(* CoDeSys 2.3.9.42 project: CR0403 AGV_25.pro *)
(* Libraries: SysLibVisu.lib 16.9.03 13:17:00, SysLibPlcCtrl.lib 13.6.03 15:49:00, SysLibFile.lib 23.9.04 10:11:36, SysLibTime.lib 27.4.05 10:36:52, SysLibTargetVisu.lib 5.4.04 13:31:00, LinuxSystemLib.Lib 18.3.03 13:26:50, ifm_CANopen\ifm_CANopen_NT_V020004.lib 3.11.15 19:07:50, ifm_pdm_file_V010006.lib 14.1.08 14:21:32, ifm_CR0403\ifm_CR0403_V030100.lib 15.1.16 15:49:16, Util.lib 6.11.07 16:39:24, ifm_J1939_NT\ifm_J1939_NT_V020004.lib 18.9.14 16:13:02, ifm_RAWCan\ifm_RAWCan_NT_V020004.lib 3.11.15 19:07:52, standard.lib 4.10.05 12:14:46, SysLibCallback.lib 26.9.08 17:43:52 *)

(* PLC configuration (modules and I/O channels)
Configuration [LocalConfiguration] node 0, in %IB0 out %QB0 {IFM_PARAM_WORD_TIME = 0}
Input/Output [LocalInputOutput] node 1, in %IB0 out %QB0
  Inputs Binary [LocalIn] node 0, in %IB0 out %QB0
    IN00 AT %IB0 [ChInputBool] Input 00 Bit
    IN01 AT %IB1 [ChInputBool] Input 01 Bit
    IN02 AT %IB2 [ChInputBool] Input 02 Bit
    IN03 AT %IB3 [ChInputBool] Input 03 Bit
    IN04 AT %IB4 [ChInputBool] Input 04 Bit
    IN05 AT %IB5 [ChInputBool] Input 05 Bit
    IN06 AT %IB6 [ChInputBool] Input 06 Bit
    IN07 AT %IB7 [ChInputBool] Input 07 Bit
    IN08 AT %IB8 [ChInputBool] Input 08 Bit
    IN09 AT %IB9 [ChInputBool] Input 09 Bit
    IN10 AT %IB10 [ChInputBool] Input 10 Bit
    IN11 AT %IB11 [ChInputBool] Input 11 Bit
  Outputs Binary [LocalOut] node 1, in %IB12 out %QB0
    OUT00 AT %QB0 [ChOutputBool] Output 00 Bit
    OUT01 AT %QB1 [ChOutputBool] Output 01 Bit
    OUT02 AT %QB2 [ChOutputBool] Output 02 Bit
    OUT03 AT %QB3 [ChOutputBool] Output 03 Bit
    OUT04 AT %QB4 [ChOutputBool] Output 04 Bit
    OUT05 AT %QB5 [ChOutputBool] Output 05 Bit
    OUT06 AT %QB6 [ChOutputBool] Output 06 Bit
    OUT07 AT %QB7 [ChOutputBool] Output 07 Bit
    OUT08 AT %QB8 [ChOutputBool] Output 08 Bit
    OUT09 AT %QB9 [ChOutputBool] Output 09 Bit
    OUT10 AT %QB10 [ChOutputBool] Output 10 Bit
    OUT11 AT %QB11 [ChOutputBool] Output 11 Bit
  System Inputs [LocalSystemInputs] node 2, in %IB12 out %QB12
    SUPPLY_VOLTAGE_VBBS AT %IW6 [ChInputWord] Supply voltage VBBS
    SUPPLY_VOLTAGE_VU AT %IW7 [ChInputWord] Supply voltage VU
    SUPPLY_VOLTAGE_VBB1 AT %IW8 [ChInputWord] Supply voltage VBB1
    SUPPLY_VOLTAGE_VBB2 AT %IW9 [ChInputWord] Supply voltage VBB2
    TEMPERATURE AT %IW10 [ChInputInt] Temperature
J1939 Interface [CAN_J1939] node 1, in %IB60 out %QB44
J1939 Interface [CAN_J1939] node 1, in %IB76 out %QB76
*)

(* Global variable list: Global_Variables *)
VAR_GLOBAL
	Route1: ARRAY [1..2,1..4] OF REAL := 10, 100, 100, 10, 10, 10, 100, 100;
	(*Route1: ARRAY [1..2,1..4] OF REAL := 10, 60, 140, 10, 10, 30, 30, 130;*)


END_VAR

VAR_GLOBAL RETAIN	(*Onze array die de aangeleerde route bevat moet een RETAIN variable zijn opdat deze zijn waarden zou blijven kennen ook bij afzetten van de spanning*)
	RouteLeren: ARRAY [1..2, 1..10] OF DWORD;
END_VAR

(* Data type *)
TYPE CONSTANTS_MATH :
STRUCT
	RadDeg : REAL := 57.29577951; (*Conversie van radialen naar degrees*)
	PI : REAL := 	3.14159265358979323846264338327950288;		(* Kreiszahl PI *)
	PI2 : REAL := 	6.28318530717958647692528676655900576;	(* PI * 2 *)
	PI4 : REAL :=  12.56637061435917295385057353311801152;	(* PI * 4 *)
	PI05 : REAL :=  1.5707963267949;							(* PI / 2 *)
	PI025 : REAL := 0.785398163397448;							(* PI / 4 *)
	PI_INV : REAL := 0.318309886183791;						(* 1 / PI *)
	E : REAL := 	2.71828182845904523536028747135266249;		(* Euler constant e *)
	E_INV : REAL := 0.367879441171442;							(* 1 / e *)
	SQ2 : REAL :=	1.4142135623731;							(* Wurzel von 2 *)
	FACTS : ARRAY[0..12] OF DINT := 1,1,2,6,24,120,720,5040,40320,362880,3628800,39916800,479001600;
END_STRUCT
END_TYPE

(* POU PLC_PRG, ST *)
PROGRAM PLC_PRG
VAR
	CAN_ENABLE_CAN2: CAN_ENABLE;
	CAN_ENABLE_CAN1: CAN_ENABLE;

	CAN_RX_ModusAGV: CAN_RX;
	Manueel: BOOL;
	Leren: BOOL;
	Automatisch: BOOL;
	UNPACK_ModusAGV: UNPACK;
	test1: BOOL;
	test2: BOOL;
END_VAR
(*Enabelen van CAN bus 1*)
CAN_ENABLE_CAN1(
	ENABLE:=TRUE ,
	CHANNEL:=1 ,
	BAUDRATE:=500 ,
	RESULT=> );

(*Enabelen van CAN bus 2 voor hetronic*)
CAN_ENABLE_CAN2(
	ENABLE:=TRUE ,
	CHANNEL:=2 ,
	BAUDRATE:=125 ,
	RESULT=> );

(*Binnenlezen modus AGV*)
CAN_RX_ModusAGV(
	ENABLE				:= TRUE,
	CHANNEL				:=1 ,
	ID						:= 16#191,
	DATA					=> ,
	RESULT				=> );

IF CAN_RX_ModusAGV.RESULT = 1
THEN
	UNPACK_ModusAGV(
	B:= CAN_RX_ModusAGV.DATA[0] ,
	B0=>Manueel ,
	B1=>Leren,
	B2=>Automatisch ,
	B3=> , 
	B4=> ,
	B5=> , 
	B6=> , 
	B7=> );
END_IF

(*Programma's die continu moeten uitgevoerd worden ongeacht de modus*)
VoedingContactor();
CAN_RX_comm_display();

(*Afhankelijk van de gewenste modus voeren we één van de onderstaande programma's uit*)
IF Manueel = TRUE
THEN
ManueleBediening();
ELSIF Leren = TRUE
THEN
AanlerenRoute();
ELSIF Automatisch = TRUE
THEN
NavSof();
END_IF
END_PROGRAM

(* POU VoedingContactor, ST *)
PROGRAM VoedingContactor
VAR

	PWM1000_Contactor_OUT7: PWM1000;
	wContactor_voeding: WORD;
	bContactor_voeding: BYTE;
END_VAR
PWM1000_Contactor_OUT7(
	ENABLE:=						TRUE ,
	CHANNEL:=					7 ,
	FREQUENCY:=				100 ,
	VALUE:=						1000 ,
	DITHER_FREQUENCY:= ,
	DITHER_VALUE:= , 
	CURRENT=>					wContactor_voeding,
	RESULT=> 					bContactor_voeding);
END_PROGRAM

(* POU CAN_RX_comm_display, ST *)
PROGRAM CAN_RX_comm_display
VAR
	CAN_RX_comm_keys_display: CAN_RX;
	UNPACK_comm_keys: UNPACK;
	keyF1: BOOL;
	keyF2: BOOL;
	keyF3: BOOL;
	keyF4: BOOL;
END_VAR
CAN_RX_comm_keys_display(
	ENABLE:=TRUE ,
	CHANNEL:=1 ,
	ID:=16#190 ,
	DATA=> ,
	RESULT=> );

IF CAN_RX_comm_keys_display.RESULT=1  THEN

UNPACK_comm_keys(
	B:=CAN_RX_comm_keys_display.DATA[0] ,
	B0=>keyF1 ,
	B1=>keyF2 ,
	B2=>keyF3,
	B3=>keyF4 ,
	B4=> ,
	B5=> , 
	B6=> , 
	B7=> );


END_IF

IF keyF1 THEN
OUT00:=TRUE;
ELSE
OUT00:=FALSE;
END_IF

IF keyF2 THEN
OUT01:=TRUE;
ELSE
OUT01:=FALSE;
END_IF
END_PROGRAM

(* POU ManueleBediening, ST *)
PROGRAM ManueleBediening
VAR
	(*Binnenlezen as1  APEM HFX*)
	INPUT_IN01_Voor_achter: INPUT;
	wVoorAchter: WORD;
	bVoorAchter: BYTE;

	(*Binnenlezen as2  APEM HFX*)
	INPUT_IN00_Links_Rechts: INPUT;
	wLinksRechts: WORD;
	bLinksRechts: BYTE;

	(*Variabele waarin de gewenste richting en snelheid wordt weggeschreven*)
	wSnelheid_ch1: DWORD := 0;
	wSnelheid_ch2: DWORD := 0;

	(*Frequentie waarop SDO write bericht verzonden wordt*)
	BLINK_SDOBericht: BLINK;
	xSDO: BOOL;

	(*SDO bericht voor channel 1 en channel 2*)
	CANOPEN_SDOWRITE_ManueleBediening_ch1: CANOPEN_SDOWRITE;
	CANOPEN_SDOWRITE_ManueleBediening_ch2: CANOPEN_SDOWRITE;
	DWORD_TO_ARRAY_ch1: DWORD_TO_ARRAY;
	DWORD_TO_ARRAY_ch2: DWORD_TO_ARRAY;

	X_as_hetronic: WORD;
	Y_as_hetronic: WORD;
	rSnelheid_ch1: REAL;
	rSnelheid_ch2: REAL;
END_VAR
(*Hier moeten we de APEM HFX binnenlezen
- Blauwe draad (verbinden we met IN01 van de CR0403:
	- Vooruit (2.5V --> 4.7V)
	- Achteruit (2.5V --> 0V)
- Gele draad (verbinden we met IN00 van de CR0403):
	- Links (2.5 --> 4.7V)
	- Rechts (2.5V --> 0V)
De switch bovenop de joystick verbindt de witte draad en de oranje draad bij indrukken
==> Deze willen we gebruiken om coördinaten op te slaan*)
(*INPUT FB om waarden as 1 joystick binnen te lezen*)
	(*INPUT_IN01_Voor_achter(
		ENABLE				:= TRUE,
		CHANNEL				:= 1,					(*We gebruiken IN01*)
		MODE					:= 3,					(*Voltage input 0 ... 10000 mV*)
		FILTER				:= ,
		VALUE					=> wVoorAchter ,		(*Bevat de spanningswaarde die we binnenlezen op IN00*)
		RESULT				=>bVoorAchter );		(*Als deze op 1 staat wil dat zeggen dat de FB is executed without error*)
(*INPUT FB om waarden as 2 joystick binnen te lezen*)
	INPUT_IN00_Links_Rechts(
		ENABLE				:= TRUE,
		CHANNEL				:= 0,					(*We gebruiken IN01*)
		MODE					:= 3,					(*Voltage input 0 ... 10000 mV*)
		FILTER				:= ,
		VALUE					=> wLinksRechts ,		(*Bevat de spanningswaarde die we binnenlezen op IN00*)
		RESULT				=>bLinksRechts );*)	(*Als deze op 1 staat wil dat zeggen dat de FB is executed without error*)

X_as_hetronic := X_as;
Y_as_hetronic := Y_as;


(*Frequentie waarop ons SDO bericht voor de roboteq aan te sturen op de bus geplaatst wordt*)
BLINK_SDOBericht(
ENABLE:= TRUE ,
TIMELOW:= t#10ms,
TIMEHIGH:=t#10ms ,
OUT=> xSDO );

(*Channel 1 Roboteq SDC2130*)
CANOPEN_SDOWRITE_ManueleBediening_ch1(
	EXECUTE				:= xSDO,
	CHANNEL				:= 1,
	NODE					:=2 ,
	IDX						:=16#2000,
	SUBIDX				:= 16#1,
	LEN					:=4 ,
	DATA					:= ,
	Timeout				:= ,
	RESULT				=> );

DWORD_TO_ARRAY_ch1(
	Word_In:=wSnelheid_ch1 ,
	P_0=>CANOPEN_SDOWRITE_ManueleBediening_ch1.DATA[0] ,
	P_1=>CANOPEN_SDOWRITE_ManueleBediening_ch1.DATA[1] ,
	P_2=>CANOPEN_SDOWRITE_ManueleBediening_ch1.DATA[2] ,
	P_3=>CANOPEN_SDOWRITE_ManueleBediening_ch1.DATA[3] );

(*Channel 2 Roboteq SDC2130*)
CANOPEN_SDOWRITE_ManueleBediening_ch2(
	EXECUTE				:= xSDO,
	CHANNEL				:= 1,
	NODE					:=2 ,
	IDX						:=16#2000,
	SUBIDX				:= 16#2,
	LEN					:=4 ,
	DATA					:= ,
	Timeout				:= ,
	RESULT				=> );

DWORD_TO_ARRAY_ch2(
	Word_In:=wSnelheid_ch2,
	P_0=>CANOPEN_SDOWRITE_ManueleBediening_ch2.DATA[0] ,
	P_1=>CANOPEN_SDOWRITE_ManueleBediening_ch2.DATA[1] ,
	P_2=>CANOPEN_SDOWRITE_ManueleBediening_ch2.DATA[2] ,
	P_3=>CANOPEN_SDOWRITE_ManueleBediening_ch2.DATA[3] );










(*VOOR_ACHTER: Vooruit en achteruit rijden*)
IF Y_as < 126 	AND X_as = 127
THEN
	(*Vooruitrijden (onderstaande commands zorgen ervoor dat onze differential drive robot rechtuit rijdt)*)
		wSnelheid_ch1 := (0+ (10*(127 - Y_as)));
		wSnelheid_ch2 := (65536 - (10*(127 - Y_as)));

ELSIF

Y_as > 128 AND X_as = 127
THEN
	(*Achteruitrijden (onderstaande commands zorgen ervoor dat onze differential drive robot rechtuit naar achter rijdt)*)
		wSnelheid_ch1 :=(65536 + (10*(127 - Y_as)));
		wSnelheid_ch2 := (0- (10*(127 - Y_as)));
ELSIF

(**)
X_as < 126 AND Y_as = 127
THEN
	(*Vooruitrijden (onderstaande commands zorgen ervoor dat onze differential drive robot rechtuit rijdt)*)
		wSnelheid_ch1 := (65536 - (10*(127 - X_as)));
		wSnelheid_ch2 := (65536 - (10*(127 - X_as)));
ELSIF

(**)
X_as > 128 AND Y_as = 127
THEN
	(*Achteruitrijden (onderstaande commands zorgen ervoor dat onze differential drive robot rechtuit naar achter rijdt)*)
		wSnelheid_ch1 := (0 - (10*(127 - X_as)));
		wSnelheid_ch2 := (0 - (10*(127 - X_as)));

ELSIF

Y_as = 127 AND X_as = 127
THEN
		wSnelheid_ch1 :=0;
		wSnelheid_ch2 :=0;
END_IF
(*

(*LINKS_RECHTS: Links en rechts rijden*)
IF wLinksRechts > 2700 AND  wVoorAchter > 2300 AND wVoorAchter <2700
THEN
	(*Links draaien*)
		wSnelheid_ch1 := (wLinksRechts - 2700)/2;
		wSnelheid_ch2 := 65536 - ((2400 - wLinksRechts)/2);

END_IF

IF wLinksRechts < 2300 AND  wVoorAchter > 2300 AND wVoorAchter <2700
THEN
	(*Rechts draaien*)
		wSnelheid_ch1 := 65536 - ((2400 - wLinksRechts)/2);
		wSnelheid_ch2 := (wLinksRechts - 2700)/2;
END_IF

(*STOPPEN: Als de joystick in het midden staat moet de AGV stoppen d.w.z. dat de ingelezen waarde zowel op de x-as als de y-as rond de 2.5V moeten zijn*)
IF wVoorAchter > 2300 AND wVoorAchter <2700 AND wLinksRechts > 2300 AND wLinksRechts <2700
THEN
	wSnelheid_ch1 := 0;
	wSnelheid_ch2 := 0;
END_IF


*)




















(*Hier moeten we de APEM HFX binnenlezen
- Blauwe draad (verbinden we met IN01 van de CR0403:
	- Vooruit (2.5V --> 4.7V)
	- Achteruit (2.5V --> 0V)
- Gele draad (verbinden we met IN00 van de CR0403):
	- Links (2.5 --> 4.7V)
	- Rechts (2.5V --> 0V)
De switch bovenop de joystick verbindt de witte draad en de oranje draad bij indrukken
==> Deze willen we gebruiken om coördinaten op te slaan*)
(*
(*Versturen cyclisch CAN bericht dat de motordata voor de Roboteq SDC2130 bevat*)
CAN_TX_ENH_CYCLIC_Roboteq(
	ENABLE				:= TRUE,
	CHANNEL				:= 1 ,
	ID						:= 16#E1 ,
	Extended				:= FALSE ,
	DataLengthCode		:= 6,
	DATA					:= ,
	PERIOD				:= t#10ms,
	RESULT				=> );

CAN_TX_ENH_CYCLIC_Roboteq.DATA[0] := bMotorDirection_ch1; (*Kan 0 of 1 bevatten en afh daarvan draait de motor CW of CCW*)
WORD_TO_ARRAY_ch1(
	Word_In				:= wSnelheid_ch1 ,
	P_0					=>CAN_TX_ENH_CYCLIC_Roboteq.DATA[1] ,
	P_1					=>CAN_TX_ENH_CYCLIC_Roboteq.DATA[2]);

CAN_TX_ENH_CYCLIC_Roboteq.DATA[3] := bMotorDirection_ch2;
WORD_TO_ARRAY_ch2(
	Word_In				:=wSnelheid_ch2,
	P_0					=>CAN_TX_ENH_CYCLIC_Roboteq.DATA[4] ,
	P_1					=>CAN_TX_ENH_CYCLIC_Roboteq.DATA[5] );

(*INPUT FB om waarden joystick binnen te lezen*)
INPUT_IN01_Voor_achter(
	ENABLE				:= TRUE,
	CHANNEL				:= 1,					(*We gebruiken IN01*)
	MODE					:= 3,					(*Voltage input 0 ... 10000 mV*)
	FILTER				:= ,
	VALUE					=> wVoorAchter ,		(*Bevat de spanningswaarde die we binnenlezen op IN00*)
	RESULT				=>bVoorAchter );		(*Als deze op 1 staat wil dat zeggen dat de FB is executed without error*)

IF wVoorAchter > 2700
THEN
	(*Vooruitrijden (onderstaande commands zorgen ervoor dat onze differential drive robot rechtuit rijdt)*)
		wVooruit := (wVoorAchter - 2700)/2;
		bMotorDirection_ch1:= 1;			(*Motor op channel 1 Roboteq draait CW*)
		wSnelheid_ch1 := wVooruit;			(*Snelheid motor op channel 1 Roboteq*)
		bMotorDirection_ch2 := 0;			(*Motor op channel 2 Roboteq draait CCW*)
		wSnelheid_ch2 := wVooruit;			(*Snelheid motor op channel 2 Roboteq*)
END_IF

IF wVoorAchter < 2400
THEN
	(*Achteruitrijden (onderstaande commands zorgen ervoor dat onze differential drive robot rechtuit naar achter rijdt)*)
		wAchter := (2400 - wVoorAchter)/2;
		bMotorDirection_ch1:= 0;			(*Motor op channel 1 Roboteq draait CW*)
		wSnelheid_ch1 := wAchter;			(*Snelheid motor op channel 1 Roboteq*)
		bMotorDirection_ch2 := 1;			(*Motor op channel 2 Roboteq draait CCW*)
		wSnelheid_ch2 := wAchter;			(*Snelheid motor op channel 2 Roboteq*)
END_IF

(*OPM: Bovenstaande dien je te herhalen indien je ook de gele draad van de joystick wilt binnenlezen*)*)
END_PROGRAM

(* POU AanlerenRoute, ST *)
PROGRAM AanlerenRoute
VAR
	xKnopRoute: BOOL;
	CAN_RX_POZXY_COORD: CAN_RX;
	ARRAY_TO_DWORD_Xcoor: ARRAY_TO_DWORD;
	ARRAY_TO_DWORD_Ycoor: ARRAY_TO_DWORD;
	xHuidigeCoordinaatCAN: DWORD;
	yHuidigeCoordinaatCAN: DWORD;
	iLeerPunt: INT := 1;
	iGrootte: INT;
	xRouteKlaar: BOOL;
	xKlaarVoorNieuweUpdate: BOOL;
	R_TRIG_AanleerModus: R_TRIG;
END_VAR
(*Telkens de drukknop van de APEM HFX joystick wordt ingedrukt
moet de huidige UWB locatie weggeschreven worden naar een ARRAY! 
Als de AGV in de 'Leren' modus zit*)
(*De drukknop verbindt de witte en oranje draad met elkaar
- Oranje draad = Vbbs CR0403
- Witte draad = IN04
*)

(*Als de drukknop op de joystick wordt ingedrukt komt de systeemvariable IN04 op TRUE te staan als de joystick is aangesloten zoals hierboven beschreven*)
xKnopRoute := IN04;

(*Binnenlezen UWB data mag continu gebeuren*)
(*Binnenlezen van de huidige positie d.m.v. UWB*)
CAN_RX_POZXY_COORD(
	ENABLE:= TRUE,
	CHANNEL:=1 ,
	ID:=16#A1 ,
	DATA=> , 
	RESULT=> );

IF  CAN_RX_POZXY_COORD.RESULT=1 THEN

ARRAY_TO_DWORD_Xcoor(
	Byte_0:=CAN_RX_POZXY_COORD.DATA[0] ,
	Byte_1:=CAN_RX_POZXY_COORD.DATA[1] ,
	Byte_2:=CAN_RX_POZXY_COORD.DATA[2] ,
	Byte_3:=CAN_RX_POZXY_COORD.DATA[3] ,
	DWORD_OUT=> xHuidigeCoordinaatCAN );

ARRAY_TO_DWORD_Ycoor(
	Byte_0:=CAN_RX_POZXY_COORD.DATA[4] ,
	Byte_1:=CAN_RX_POZXY_COORD.DATA[5] ,
	Byte_2:=CAN_RX_POZXY_COORD.DATA[6] ,
	Byte_3:=CAN_RX_POZXY_COORD.DATA[7] ,
	DWORD_OUT=> yHuidigeCoordinaatCAN );
END_IF
(*Elke keer er op de drukknop gedrukt wordt moet de huidige UWB coördinaat weggeschreven worden naar een array
IF xKnopRoute = TRUE
THEN
Route1[1,i_EindPunt];*)
(*Ervoor zorgen dat er maar één keer per indrukken van de joystick, een update van de array doen*)
(*IF xKnopRoute = FALSE
THEN
xKlaarVoorNieuweUpdate := TRUE;
ELSE
xKlaarVoorNieuweUpdate := FALSE;
END_IF*)

R_TRIG_AanleerModus(
CLK			:=  xKnopRoute,
Q				=> xKlaarVoorNieuweUpdate );

(*IF structuur dat indien drukknop joystick ingedrukt wordt de huidge UWB locatie weggeschreven wordt naar de array RouteLeren*)
IF xKlaarVoorNieuweUpdate = TRUE AND xRouteKlaar = FALSE
THEN
RouteLeren[1, iLeerPunt] := xHuidigeCoordinaatCAN;
RouteLeren[2, iLeerPunt] := yHuidigeCoordinaatCAN;
iLeerPunt := iLeerPunt + 1;


iGrootte := SIZEOF(RouteLeren)/8;

		IF iGrootte < iLeerPunt
		THEN
		xRouteKlaar := TRUE;
		ELSE
		xRouteKlaar := FALSE;
		END_IF
END_IF

(*Can bericht versturen naar het scherm over welke welk punt van de route dat we reeds zitten en of het laatste punt van de aangeleerde route bereikt is*)
(*Toekomstmuziek dat doorsturen naar de CR0451*)
END_PROGRAM

(* POU NavSof, ST *)
PROGRAM NavSof
VAR
	(*Variabelen voor het binnen lezen van de UWB data via de CAN bus*)
	CAN_RX_POZXY_COORD: CAN_RX;							(*FB om een CAN bericht binnen te lezen*)
	ARRAY_TO_DWORD_Xcoor: ARRAY_TO_DWORD;				(*Data van een ARRAY naar een getal omvormen*)
	xHuidigeCoordinaat: REAL;										(*Datatype vastleggen*)
	ARRAY_TO_DWORD_Ycoor: ARRAY_TO_DWORD;
	yHuidigeCoordinaat: REAL;

	(*Variabelen NavSof*)
	i_Waypoints: INT := 0;													(*Variabele die het aantal waypoints van onze huidige route bevat*)
	x_Jumplock: BOOL := TRUE;											(*Flag zodat bij opstart éénmalig X en Y-huidig kunnen gebruikt worden als X en Y start voor de trackline*)
	xStartCoordinaat: REAL := 0;											(*X coordinaat voor begin trackline*)
	yStartCoordinaat: REAL := 0;											(*Y coordinaat voor einde trackline*)
	xEindCoordinaat: REAL := 0;											(*X coordinaat voor einde trackline*)
	yEindCoordinaat: REAL := 0;											(*Y coordinaat voor einde trackline*)
	rAfstandTotWaypoint: REAL := 0;										(*Bevat de afstand tot het waypoint*)
	rTrackHoek: REAL:= 0;												(*Bevat de trackhoek, de hoek die de AGV naar links of rechts doet sturen opdat deze terug op de trackline zou uitkomen*)
	CONSTANTS_MATH: CONSTANTS_MATH;							(*Struct die bepaalde wiskundige constanten bevat*)


	rHoekAGV: REAL;
	rTrack: REAL;
	BNO_lock: BOOL;
	StuurLinks: REAL;
	beginBNO: REAL;
	eindeBNO: REAL;
	StuurNeutraal: REAL;
	StuurRechts: REAL;
	rAfstandEncoder: REAL;
	VooruitRijden: REAL;
	Stoppen: REAL;
	i_EindPunt: INT:=1;
	i_StartPunt: INT:=1;
	CAN_RX_BNO: CAN_RX;
	ARRAY_TO_DWORD_BNO: ARRAY_TO_DWORD;
	OrientatieAGV: REAL;
	BNO_jumplock: BOOL;
	dot: REAL;
	det: REAL;
	angle: REAL;
	Encoder_jumplock: BOOL;
	beginEncoderLinks: REAL;
	beginEncoderRechts: REAL;
	UWB_jumplock: BOOL := TRUE;
	xHuidigeCoordinaatCAN: REAL;
	yHuidigeCoordinaatCAN: REAL;
	START_jumplock: BOOL;
	xIni: BOOL;
	rHoekVorigAGV: REAL;
	dot_wp: REAL;
	det_wp: REAL;
	angle_wp: REAL;
	rotate_angle: REAL;
	Rotatie_Rechts_wp: Rotatie;
	Rechts_ok: BOOL;
	Rotatie_Links_wp: Rotatie;
	Links_ok: BOOL;
	Rotatie_Links: Rotatie;
	HoekLinks: BOOL;
	HoekRechts: BOOL;
	iControl: INT := 120; (*iControl een waarde geven verschillend van 0 zodat wij bepalen wnr de initialisatie gestart wordt!*)
	Links: INT;
	Rechts: INT;
	CAN_TX_ENH_CYCLIC_Roboteq: CAN_TX_ENH_CYCLIC;
	bMotorDirection_ch1: BYTE;
	WORD_TO_ARRAY_ch1: WORD_TO_ARRAY;
	wSnelheid_ch1: WORD;
	bMotorDirection_ch2: BYTE;
	WORD_TO_ARRAY_ch2: WORD_TO_ARRAY;
	wSnelheid_ch2: WORD;
	OrientatieAGV_deg: DWORD;
	rHoekAGV_rad: REAL;
	VerdraaiingTotVolgendeWaypoint: REAL;
END_VAR
(*Binnenlezen van de huidige positie d.m.v. UWB*)
CAN_RX_POZXY_COORD(
	ENABLE:= TRUE,
	CHANNEL:=1 ,
	ID:=16#A1 ,
	DATA=> , 
	RESULT=> );

IF  CAN_RX_POZXY_COORD.RESULT=1 THEN

ARRAY_TO_DWORD_Xcoor(
	Byte_0:=CAN_RX_POZXY_COORD.DATA[0] ,
	Byte_1:=CAN_RX_POZXY_COORD.DATA[1] ,
	Byte_2:=CAN_RX_POZXY_COORD.DATA[2] ,
	Byte_3:=CAN_RX_POZXY_COORD.DATA[3] ,
	DWORD_OUT=> xHuidigeCoordinaatCAN );

ARRAY_TO_DWORD_Ycoor(
	Byte_0:=CAN_RX_POZXY_COORD.DATA[4] ,
	Byte_1:=CAN_RX_POZXY_COORD.DATA[5] ,
	Byte_2:=CAN_RX_POZXY_COORD.DATA[6] ,
	Byte_3:=CAN_RX_POZXY_COORD.DATA[7] ,
	DWORD_OUT=> yHuidigeCoordinaatCAN );
END_IF

(*Versturen cyclisch CAN bericht dat de motordata voor de Roboteq SDC2130 controller bevat*)
CAN_TX_ENH_CYCLIC_Roboteq(
	ENABLE				:= TRUE ,
	CHANNEL				:= 1 ,
	ID						:= 16#E1 ,
	Extended				:= FALSE ,
	DataLengthCode		:= 6 ,
	DATA					:= ,
	PERIOD				:= t#10ms ,
	RESULT				=> );

CAN_TX_ENH_CYCLIC_Roboteq.DATA[0] := bMotorDirection_ch1; (*Kan 0 of 1 bevatten en afh daarvan draait de motor CW of CCW*)
WORD_TO_ARRAY_ch1(
	Word_In				:= wSnelheid_ch1 ,
	P_0					=>CAN_TX_ENH_CYCLIC_Roboteq.DATA[1] ,
	P_1					=>CAN_TX_ENH_CYCLIC_Roboteq.DATA[2]);

CAN_TX_ENH_CYCLIC_Roboteq.DATA[3] := bMotorDirection_ch2;
WORD_TO_ARRAY_ch2(
	Word_In				:=wSnelheid_ch2,
	P_0					=>CAN_TX_ENH_CYCLIC_Roboteq.DATA[4] ,
	P_1					=>CAN_TX_ENH_CYCLIC_Roboteq.DATA[5] );


(*Ervoor zorgen dat we pas een UWB update krijgen bij aankomst aan ons volgende waypoint*)
IF UWB_jumplock = TRUE
THEN
	yHuidigeCoordinaat := yHuidigeCoordinaatCAN;
	xHuidigeCoordinaat := xHuidigeCoordinaatCAN;
	IF (xHuidigeCoordinaat = 0 AND yHuidigeCoordinaat = 0)
	THEN
	UWB_jumplock := TRUE;
	ELSE
	UWB_jumplock := FALSE;
	END_IF
END_IF;

(*Het aantal waypoints van onze huidige route bepalen*)
i_Waypoints := SIZEOF(Route1)/8;							(*Route 1 bevat 2 * 4 coordinaten die telkens 4 bytes (datatype REAL) innemen
																de totale grootte van deze array is dus 32 bytes / 8 geeft ons het aantal waypoints*)

(*Ervoor zorgen dat bij opstart éénmalig X- en Y-huidig gebruikt kunnen worden als X- en Y-start voor de trackline*)
IF( x_Jumplock = TRUE AND UWB_jumplock = FALSE)
THEN
	xStartCoordinaat := xHuidigeCoordinaat;
	yStartCoordinaat := yHuidigeCoordinaat;
	x_Jumplock := FALSE;
	iControl := 0; 												(*Hier gaan we over naar de initialisatie fase*)
END_IF;

(*xEindCoordinaat en yEindcoordinaat halen we uit een ARRAY*)
xEindCoordinaat := Route1[1,i_EindPunt];
yEindCoordinaat := Route1[2,i_EindPunt];

(*Ervoor zorgen dat bij het afleggen van een route er steeds geweten is of je links of rechts van je trackline zit
Vervolgens moet de AGV een gegeven hoek naar links of rechts verdraaien en daarnaa rechtuit rijden*)
(*Mogen we pas berekenen als UWB_ lock = FALSE staat!*)
IF (x_Jumplock = FALSE AND UWB_jumplock = FALSE)
THEN
	IF xStartCoordinaat > xEindCoordinaat OR yStartCoordinaat > yEindCoordinaat
	THEN
	rTrack := ATAN2(  yStartCoordinaat - yEindCoordinaat  ,  xStartCoordinaat -  xEindCoordinaat)*57.29577951;
	rHoekAGV := ATAN2( yHuidigeCoordinaat - yEindCoordinaat  ,   xHuidigeCoordinaat - xEindCoordinaat )*57.29577951;
	ELSE
	rTrack := ATAN2(yEindCoordinaat - yStartCoordinaat  ,  xEindCoordinaat - xStartCoordinaat)*57.29577951;
	rHoekAGV := ATAN2(yEindCoordinaat - yHuidigeCoordinaat ,  xEindCoordinaat - xHuidigeCoordinaat )*57.29577951;
	END_IF

END_IF;

(*Implementatie van een stappensturing in de software*)
CASE iControl OF				(*In deze stappen vindt men handelingen terug die niet gelijktijdig uitgevoerd mogen worden*)
0: (*Initialisatiefase*)(*Initialisatie AGV zodat zijn oriëntatie in het UWB x/y-assenstelsel kan bepaald worden*)
		IF Encoder_jumplock = TRUE												(*De variabele beginEncoder mag enkel upgedate worden met de huidige Encoder waarde bij verspringen van waypoint!*)
		THEN
		beginEncoderLinks:= PosEncoderLinks;										(*Hierin moet de waarde van de encoder opgeslaan worden, deze waarde mag niet meer upgedate worden tot het volgende waypoint bereikt is*)
		beginEncoderRechts := PosEncoderRechts;
		Encoder_jumplock := FALSE;											(*Ervoor zorgen dat de variabele beginEncoder niet meer wordt aangepast zolang er niet van waypoint versprongen is*)
		END_IF
		IF 30> ABS(PosEncoderLinks - beginEncoderLinks)				(*Bedoeling het programma blijft hier hangen tot dit stukje code is uitgevoerd, het kan enkel onderbroken worden door de veiligheidssensoren*)
		THEN
		(*Vooruitrijden (onderstaande commands zorgen ervoor dat onze differential drive robot rechtuit rijdt)*)
		bMotorDirection_ch1:= 1;			(*Motor op channel 1 Roboteq draait CW*)
		wSnelheid_ch1 := 150;			(*Snelheid motor op channel 1 Roboteq*)
		bMotorDirection_ch2 := 0;			(*Motor op channel 2 Roboteq draait CCW*)
		wSnelheid_ch2 := 150;			(*Snelheid motor op channel 2 Roboteq*)
		ELSE
		(*Stoppen (onderstaande commands zorgen ervoor dat onze differential drive robot stopt)*)
		bMotorDirection_ch1:= 1;			(*Motor op channel 1 Roboteq draait CW*)
		wSnelheid_ch1 := 0;				(*Snelheid motor op channel 1 Roboteq*)
		bMotorDirection_ch2 := 0;			(*Motor op channel 2 Roboteq draait CCW*)
		wSnelheid_ch2 := 0;				(*Snelheid motor op channel 2 Roboteq*)

		Encoder_jumplock := TRUE;
		UWB_jumplock := TRUE;													(*Na het afronden van de initialisatie dienen we opnieuw een update te krijgen van waar we zijn m.b.v. UWB, daarom plaatsen we het UWB_lock op TRUE*)
		iControl := 1;
		END_IF
1: (*Bepalen of de AGV naar links of rechts moet draaien*)
		IF rTrack < rHoekAGV														(*Onder deze voorwaarde zitten we rechts van onze trackline en moeten we dus naar links sturen*)
		THEN
				iControl := 2;														(*Links draaien*)

		ELSIF rTrack > rHoekAGV
		THEN
				iControl := 3;														(*Rechts draaien*)
		END_IF;

2: (*LinksDraaien*)
		(*Binnenlezen orientatie afkomstig van de BNO055*)
		CAN_RX_BNO(
			ENABLE:= TRUE,
			CHANNEL:=1 ,
			ID:=16#B1 ,
			DATA=> ,
			RESULT=> );

		IF  CAN_RX_BNO.RESULT=1 THEN

		ARRAY_TO_DWORD_BNO(
			Byte_0:=CAN_RX_BNO.DATA[0] ,
			Byte_1:=CAN_RX_BNO.DATA[1] ,
			Byte_2:=CAN_RX_BNO.DATA[2] ,
			Byte_3:=CAN_RX_BNO.DATA[3] ,
			DWORD_OUT=> OrientatieAGV_deg );
		END_IF

		OrientatieAGV := (OrientatieAGV_deg * CONSTANTS_MATH.PI) / 180; (*De COS, SIN ... in ST verwachten een argument in rad ipv deg daarom moet onze deg omgerekend worden naar rad*)

		IF BNO_jumplock = TRUE										(*De variabele beginBNO mag enkel upgedate worden met de huidige BNO waarde bij verspringen van waypoint!*)
		THEN
		beginBNO:= OrientatieAGV;										(*Hierin moet de waarde van de BNO055 opgeslaan worden, deze waarde mag niet meer upgedate worden tot het volgende waypoint bereikt is*)
		BNO_jumplock := FALSE;											(*Ervoor zorgen dat de variabele beginBNO niet meer wordt aangepast zolang er niet van waypoint versprongen is*)
		END_IF

		(*Onderstaande code moet ervoor zorgen dat er steeds de clockwise hoek tussen de twee vectoren berekent wordt!*)
		dot := (COS(beginBNO)*COS(OrientatieAGV))+(SIN(beginBNO)*SIN(OrientatieAGV));
		det := (COS(beginBNO)*SIN(OrientatieAGV)) - (SIN(beginBNO)*COS(OrientatieAGV));
		angle := (ATAN2(det, dot))*57.29577951;

		IF  ABS(rTrack-rHoekAGV)> ABS(angle)
		THEN
		(*Links draaien (onderstaande commands zorgen ervoor dat onze differential drive robot links draait)*)
		bMotorDirection_ch1:= 1;			(*Motor op channel 1 Roboteq draait CW*)
		wSnelheid_ch1 := 200;			(*Snelheid motor op channel 1 Roboteq*)
		bMotorDirection_ch2 := 1;			(*Motor op channel 2 Roboteq draait CCW*)
		wSnelheid_ch2 := 200;			(*Snelheid motor op channel 2 Roboteq*)
		ELSE
		(*Stoppen/ stuurneutraal (onderstaande commands zorgen ervoor dat onze differential drive robot stopt)*)
		bMotorDirection_ch1:= 1;			(*Motor op channel 1 Roboteq draait CW*)
		wSnelheid_ch1 := 0;				(*Snelheid motor op channel 1 Roboteq*)
		bMotorDirection_ch2 := 0;			(*Motor op channel 2 Roboteq draait CCW*)
		wSnelheid_ch2 := 0;				(*Snelheid motor op channel 2 Roboteq*)

		BNO_jumplock := TRUE;
		iControl := 4;
		END_IF
3: (*RechtsDraaien*)
		(*Binnenlezen orientatie afkomstig van de BNO055*)
		CAN_RX_BNO(
			ENABLE:= TRUE,
			CHANNEL:=1 ,
			ID:=16#B1 ,
			DATA=> ,
			RESULT=> );

		IF  CAN_RX_BNO.RESULT=1 THEN

		ARRAY_TO_DWORD_BNO(
			Byte_0:=CAN_RX_BNO.DATA[0] ,
			Byte_1:=CAN_RX_BNO.DATA[1] ,
			Byte_2:=CAN_RX_BNO.DATA[2] ,
			Byte_3:=CAN_RX_BNO.DATA[3] ,
			DWORD_OUT=> OrientatieAGV_deg );
		END_IF

		OrientatieAGV := (OrientatieAGV_deg * CONSTANTS_MATH.PI) / 180; (*De COS, SIN ... in ST verwachten een argument in rad ipv deg daarom moet onze deg omgerekend worden naar rad*)


		IF BNO_jumplock = TRUE										(*De variabele beginBNO mag enkel upgedate worden met de huidige BNO waarde bij verspringen van waypoint!*)
		THEN
		beginBNO:= OrientatieAGV;										(*Hierin moet de waarde van de BNO055 opgeslaan worden, deze waarde mag niet meer upgedate worden tot het volgende waypoint bereikt is*)
		BNO_jumplock := FALSE;											(*Ervoor zorgen dat de variabele beginBNO niet meer wordt aangepast zolang er niet van waypoint versprongen is*)
		END_IF

		(*Onderstaande code moet ervoor zorgen dat er steeds de clockwise hoek tussen de twee vectoren berekent wordt!*)
		dot := (COS(beginBNO)*COS(OrientatieAGV))+(SIN(beginBNO)*SIN(OrientatieAGV));
		det := (COS(beginBNO)*SIN(OrientatieAGV)) - (SIN(beginBNO)*COS(OrientatieAGV));
		angle := (ATAN2(det, dot))*57.29577951;

		IF  ABS(rTrack-rHoekAGV)> ABS(angle)
		THEN
		(*Rechts draaien (onderstaande commands zorgen ervoor dat onze differential drive robot links draait)*)
		bMotorDirection_ch1:= 0;			(*Motor op channel 1 Roboteq draait CW*)
		wSnelheid_ch1 := 200;			(*Snelheid motor op channel 1 Roboteq*)
		bMotorDirection_ch2 := 0;			(*Motor op channel 2 Roboteq draait CCW*)
		wSnelheid_ch2 := 200;			(*Snelheid motor op channel 2 Roboteq*)
		ELSE
		(*Stoppen/ stuurneutraal (onderstaande commands zorgen ervoor dat onze differential drive robot stopt)*)
		bMotorDirection_ch1:= 1;			(*Motor op channel 1 Roboteq draait CW*)
		wSnelheid_ch1 := 0;				(*Snelheid motor op channel 1 Roboteq*)
		bMotorDirection_ch2 := 0;			(*Motor op channel 2 Roboteq draait CCW*)
		wSnelheid_ch2 := 0;				(*Snelheid motor op channel 2 Roboteq*)

		BNO_jumplock := TRUE;
		iControl := 4;
		END_IF
4: (*StuurNeutraal en rechtdoor rijden tot wanneer het waypoint bereikt is*)
		(*Uitrekenen wat de afstand tot het volgende waypoint is*)
		rAfstandTotWaypoint := Afstand_Punt_Punt(xStartCoordinaat, yStartCoordinaat, xEindCoordinaat, yEindCoordinaat);

		(*De richting is reeds gekend, de afstand tot het volgende waypoint ook, nu moeten we de robot vooruit laten rijden tot het volgende waypoint
		Merk op het is enkel de encoder langs de kant waarbij niet gedraaid wordt die de correcte afstand zal weergeven!*)
		IF Encoder_jumplock = TRUE												(*De variabele beginEncoder mag enkel upgedate worden met de huidige Encoder waarde bij verspringen van waypoint!*)
		THEN
		beginEncoderLinks:= PosEncoderLinks;										(*Hierin moet de waarde van de encoder opgeslaan worden, deze waarde mag niet meer upgedate worden tot het volgende waypoint bereikt is*)
		beginEncoderRechts := PosEncoderRechts;
		Encoder_jumplock := FALSE;											(*Ervoor zorgen dat de variabele beginEncoder niet meer wordt aangepast zolang er niet van waypoint versprongen is*)
		END_IF


		IF rAfstandTotWaypoint>= ((PosEncoderLinks-beginEncoderLinks) + (PosEncoderRechts - beginEncoderRechts))/2
		THEN
		(*Vooruitrijden (onderstaande commands zorgen ervoor dat onze differential drive robot rechtuit rijdt)*)
		bMotorDirection_ch1:= 1;			(*Motor op channel 1 Roboteq draait CW*)
		wSnelheid_ch1 := 400;			(*Snelheid motor op channel 1 Roboteq*)
		bMotorDirection_ch2 := 0;			(*Motor op channel 2 Roboteq draait CCW*)
		wSnelheid_ch2 := 400;			(*Snelheid motor op channel 2 Roboteq*)
		ELSE
		(*Stoppen (onderstaande commands zorgen ervoor dat onze differential drive robot stopt)*)
		bMotorDirection_ch1:= 1;			(*Motor op channel 1 Roboteq draait CW*)
		wSnelheid_ch1 := 0;				(*Snelheid motor op channel 1 Roboteq*)
		bMotorDirection_ch2 := 0;			(*Motor op channel 2 Roboteq draait CCW*)
		wSnelheid_ch2 := 0;				(*Snelheid motor op channel 2 Roboteq*)

		i_StartPunt := i_EindPunt;
		xStartCoordinaat := Route1[1,i_StartPunt];
		yStartCoordinaat := Route1[2,i_StartPunt];
		i_EindPunt := i_EindPunt +1;

		IF i_EindPunt > i_Waypoints								(*Ervoor zorgen dat we steeds opnieuw onze route kunnen afleggen door de index van de array te resetten als het laatste waypoint bereikt is! *)
		THEN
		i_EindPunt:= 1;
		END_IF;

				(*xEindCoordinaat en yEindcoorinaat halen we uit een ARRAY*)
				xEindCoordinaat := Route1[1,i_EindPunt];
				yEindCoordinaat := Route1[2,i_EindPunt];

				(*Aangekomen op het waypoint moeten we draaien naar het volgende waypoint!*)
				(*Daarvoor dienen we steeds de clockwise hoek te bepalen tussen de vector HoekVorigAGV en de vector rTrack*)

				rHoekVorigAGV := (rHoekAGV* CONSTANTS_MATH.PI) / 180;

				iControl := 5; (*Laten uitrekenen of er naar links of rechts moet gedraaid worden en hoeveel er moet gedraaid worden*)
		END_IF
5: (*Bepalen of er bij bereiken waypoint naar links of rechts gedraaid moet worden om het andere waypoint te bereiken, en ook hoeveel er dan moet gedraaid worden*)

(*Onderstaande code moet ervoor zorgen dat er steeds de clockwise hoek tussen de twee vectoren berekent wordt!*)
				rHoekAGV_rad := (ATAN2(yEindCoordinaat - yStartCoordinaat  ,  xEindCoordinaat - xStartCoordinaat)* CONSTANTS_MATH.PI) / 180; (*NOg verieferen of dit altijd klopt!*)

				dot := (COS(rHoekVorigAGV)*COS(rHoekAGV_rad))+(SIN(rHoekVorigAGV)*SIN(rHoekAGV_rad));
				det := (COS(rHoekVorigAGV)*SIN(rHoekAGV_rad)) - (SIN(rHoekVorigAGV)*COS(rHoekAGV));
				VerdraaiingTotVolgendeWaypoint := (ATAN2(det, dot))*57.29577951;
				(*Onderstaande code moet ervoor zorgen dat we op een waypoint ons juist orienteren tot het volgende waypoint*)
				(*rTrack := ATAN2(yStartCoordinaat - yEindCoordinaat , xStartCoordinaat -  xEindCoordinaat )*57.29577951;
				rHoekVorigAGV := rHoekAGV;*)



				(*Nu moeten we deze hoek naar links of naar rechts draaien of niets doen, als hij juist georiënteerd staat*)

				IF VerdraaiingTotVolgendeWaypoint > 0
				THEN
						iControl := 6;
				ELSIF VerdraaiingTotVolgendeWaypoint < 0
				THEN
						iControl := 7;
				ELSE
						iControl := 1;
				END_IF;
6: (*Oorspronkelijke verdraaiing opheffen => LinksDraaien*)
		(*Binnenlezen orientatie afkomstig van de BNO055*)
		CAN_RX_BNO(
			ENABLE:= TRUE,
			CHANNEL:=1 ,
			ID:=16#B1 ,
			DATA=> ,
			RESULT=> );

		IF  CAN_RX_BNO.RESULT=1 THEN

		ARRAY_TO_DWORD_BNO(
			Byte_0:=CAN_RX_BNO.DATA[0] ,
			Byte_1:=CAN_RX_BNO.DATA[1] ,
			Byte_2:=CAN_RX_BNO.DATA[2] ,
			Byte_3:=CAN_RX_BNO.DATA[3] ,
			DWORD_OUT=> OrientatieAGV_deg );
		END_IF

		OrientatieAGV := (OrientatieAGV_deg * CONSTANTS_MATH.PI) / 180; (*De COS, SIN ... in ST verwachten een argument in rad ipv deg daarom moet onze deg omgerekend worden naar rad*)


		IF BNO_jumplock = TRUE										(*De variabele beginBNO mag enkel upgedate worden met de huidige BNO waarde bij verspringen van waypoint!*)
		THEN
		beginBNO:= OrientatieAGV;										(*Hierin moet de waarde van de BNO055 opgeslaan worden, deze waarde mag niet meer upgedate worden tot het volgende waypoint bereikt is*)
		BNO_jumplock := FALSE;											(*Ervoor zorgen dat de variabele beginBNO niet meer wordt aangepast zolang er niet van waypoint versprongen is*)
		END_IF

		(*Onderstaande code moet ervoor zorgen dat er steeds de clockwise hoek tussen de twee vectoren berekent wordt!*)
		dot := (COS(beginBNO)*COS(OrientatieAGV))+(SIN(beginBNO)*SIN(OrientatieAGV));
		det := (COS(beginBNO)*SIN(OrientatieAGV)) - (SIN(beginBNO)*COS(OrientatieAGV));
		angle := (ATAN2(det, dot))*57.29577951;

		IF  ABS(rTrack - rHoekVorigAGV)> ABS(angle)
		THEN
		(*Links draaien (onderstaande commands zorgen ervoor dat onze differential drive robot links draait)*)
		bMotorDirection_ch1:= 1;			(*Motor op channel 1 Roboteq draait CW*)
		wSnelheid_ch1 := 200;			(*Snelheid motor op channel 1 Roboteq*)
		bMotorDirection_ch2 := 1;			(*Motor op channel 2 Roboteq draait CCW*)
		wSnelheid_ch2 := 200;			(*Snelheid motor op channel 2 Roboteq*)
		ELSE
		(*Stoppen/ stuurneutraal (onderstaande commands zorgen ervoor dat onze differential drive robot stopt)*)
		bMotorDirection_ch1:= 1;			(*Motor op channel 1 Roboteq draait CW*)
		wSnelheid_ch1 := 0;				(*Snelheid motor op channel 1 Roboteq*)
		bMotorDirection_ch2 := 0;			(*Motor op channel 2 Roboteq draait CCW*)
		wSnelheid_ch2 := 0;				(*Snelheid motor op channel 2 Roboteq*)

		BNO_jumplock := TRUE;
		UWB_jumplock := TRUE;											(*Ervoor zorgen dat we terug een UWB update krijgen*)
		iControl := 1;
		END_IF
7: (*Oorspronkelijke verdraaiing opheffen => RechtsDraaien*)
		(*Binnenlezen orientatie afkomstig van de BNO055*)
		CAN_RX_BNO(
			ENABLE:= TRUE,
			CHANNEL:=1 ,
			ID:=16#B1 ,
			DATA=> ,
			RESULT=> );

		IF  CAN_RX_BNO.RESULT=1 THEN

		ARRAY_TO_DWORD_BNO(
			Byte_0:=CAN_RX_BNO.DATA[0] ,
			Byte_1:=CAN_RX_BNO.DATA[1] ,
			Byte_2:=CAN_RX_BNO.DATA[2] ,
			Byte_3:=CAN_RX_BNO.DATA[3] ,
			DWORD_OUT=> OrientatieAGV_deg );
		END_IF

		OrientatieAGV := (OrientatieAGV_deg * CONSTANTS_MATH.PI) / 180; (*De COS, SIN ... in ST verwachten een argument in rad ipv deg daarom moet onze deg omgerekend worden naar rad*)


		IF BNO_jumplock = TRUE										(*De variabele beginBNO mag enkel upgedate worden met de huidige BNO waarde bij verspringen van waypoint!*)
		THEN
		beginBNO:= OrientatieAGV;										(*Hierin moet de waarde van de BNO055 opgeslaan worden, deze waarde mag niet meer upgedate worden tot het volgende waypoint bereikt is*)
		BNO_jumplock := FALSE;											(*Ervoor zorgen dat de variabele beginBNO niet meer wordt aangepast zolang er niet van waypoint versprongen is*)
		END_IF

		(*Onderstaande code moet ervoor zorgen dat er steeds de clockwise hoek tussen de twee vectoren berekent wordt!*)
		dot := (COS(beginBNO)*COS(OrientatieAGV))+(SIN(beginBNO)*SIN(OrientatieAGV));
		det := (COS(beginBNO)*SIN(OrientatieAGV)) - (SIN(beginBNO)*COS(OrientatieAGV));
		angle := (ATAN2(det, dot))*57.29577951;

		IF  ABS(rTrack - rHoekVorigAGV)> ABS(angle)
		THEN
		(*Rechts draaien (onderstaande commands zorgen ervoor dat onze differential drive robot links draait)*)
		bMotorDirection_ch1:= 0;			(*Motor op channel 1 Roboteq draait CW*)
		wSnelheid_ch1 := 200;			(*Snelheid motor op channel 1 Roboteq*)
		bMotorDirection_ch2 := 0;			(*Motor op channel 2 Roboteq draait CCW*)
		wSnelheid_ch2 := 200;			(*Snelheid motor op channel 2 Roboteq*)
		ELSE
		(*Stoppen/ stuurneutraal (onderstaande commands zorgen ervoor dat onze differential drive robot stopt)*)
		bMotorDirection_ch1:= 1;			(*Motor op channel 1 Roboteq draait CW*)
		wSnelheid_ch1 := 0;				(*Snelheid motor op channel 1 Roboteq*)
		bMotorDirection_ch2 := 0;			(*Motor op channel 2 Roboteq draait CCW*)
		wSnelheid_ch2 := 0;				(*Snelheid motor op channel 2 Roboteq*)

		BNO_jumplock := TRUE;
		UWB_jumplock := TRUE;											(*Ervoor zorgen dat we terug een UWB update krijgen*)
		iControl := 1;
		END_IF
END_CASE
END_PROGRAM

(* POU FBNavSof/Rotatie, ST *)
FUNCTION_BLOCK Rotatie
VAR_INPUT
	GewensteHoekVerdraaiing: REAL;
	Richting: BOOL;
END_VAR
VAR_OUTPUT
	HoekOk: BOOL;
END_VAR
VAR
	CAN_RX_BNO: CAN_RX;
	OrientatieAGV: REAL;
	ARRAY_TO_DWORD_BNO: ARRAY_TO_DWORD;
	beginBNO: REAL;
	BNO_jumplock: BOOL;
	dot: REAL;
	det: REAL;
	angle: REAL;
	Rechts: REAL;
	Links: REAL;
END_VAR
(******
Doel: In de juiste richting (links of rechts) een ingegeven hoek verdraaiien.
Input:
rreal hoek
boolean (rechts is TRUE en links is FALSE)
Output: boolean
*****)

GewensteHoekVerdraaiing;											(*Waarde tussen 0 en 360° *)
Richting;																(*True = Rechts en False = Links*)
HoekOk;																(*Boolean die*)

(*Binnenlezen orientatie afkomstig van de BNO055*)
CAN_RX_BNO(
	ENABLE:= TRUE,
	CHANNEL:=1 ,
	ID:=16#B1 ,
	DATA=> , 
	RESULT=> );

IF  CAN_RX_BNO.RESULT=1 THEN

ARRAY_TO_DWORD_BNO(
	Byte_0:=CAN_RX_BNO.DATA[0] ,
	Byte_1:=CAN_RX_BNO.DATA[1] ,
	Byte_2:=CAN_RX_BNO.DATA[2] ,
	Byte_3:=CAN_RX_BNO.DATA[3] ,
	DWORD_OUT=> OrientatieAGV );

END_IF


IF BNO_jumplock = TRUE										(*De variabele beginBNO mag enkel upgedate worden met de huidige BNO waarde bij verspringen van waypoint!*)
THEN
beginBNO:= OrientatieAGV;										(*Hierin moet de waarde van de BNO055 opgeslaan worden, deze waarde mag niet meer upgedate worden tot het volgende waypoint bereikt is*)
BNO_jumplock := FALSE;											(*Ervoor zorgen dat de variabele beginBNO niet meer wordt aangepast zolang er niet van waypoint versprongen is*)
END_IF

(*Onderstaande code moet ervoor zorgen dat er steeds de clockwise hoek tussen de twee vectoren berekent wordt!*)
dot := (COS(beginBNO)*COS(OrientatieAGV))+(SIN(beginBNO)*SIN(OrientatieAGV));
det := (COS(beginBNO)*SIN(OrientatieAGV)) - (SIN(beginBNO)*COS(OrientatieAGV));
angle := (ATAN2(det, dot))*57.29577951;

IF GewensteHoekVerdraaiing > ABS(angle)
THEN
	IF Richting = TRUE
	THEN
	Rechts; 														(*Hier moet het commando komen zodat de Roboteq de rechtermotor aanstuurt en de linkermotor niet aanstuurt*)
	ELSIF Richting = FALSE
	THEN
	Links;															(*Hier moet het commando komen zodat de Roboteq de linkermotor aanstuurt en de rechtermotor niet aanstuurt*)
	END_IF;
	HoekOk := FALSE;
ELSE
	HoekOk := TRUE;
END_IF;
END_FUNCTION_BLOCK

(* POU FunctiesNavSof/ATAN2, ST *)
FUNCTION ATAN2 : REAL
VAR_INPUT
	Y : REAL;
	X : REAL;
END_VAR
VAR
	MATH: CONSTANTS_MATH;
END_VAR
IF X > 0.0 THEN
	ATAN2 := ATAN(Y/X);
ELSIF X < 0.0 THEN
	IF Y >=0.0 THEN
		ATAN2 := ATAN(Y/X) + MATH.PI;
	ELSE
		ATAN2 := ATAN(Y/X) - MATH.PI;
	END_IF;
ELSIF Y > 0.0 THEN
	ATAN2 := MATH.PI05;
ELSIF Y < 0.0 THEN
	ATAN2 := -MATH.PI05;
ELSE
	ATAN2 := 0.0;
END_IF;




(* revision history hm	20.  apr. 2008	rev 1.0 original version
hm	18. oct. 2008	rev 1.1 	changed to use math constants
hm	10. mar. 2009	rev 1.2	real constants updated to new systax using dot
*)
END_FUNCTION

(* POU FunctiesNavSof/Afstand_Punt_Punt, ST *)
FUNCTION Afstand_Punt_Punt : REAL
VAR_INPUT
	X1 : REAL;
	Y1 : REAL;
	X2 : REAL;
	Y2 : REAL;
END_VAR
VAR
END_VAR
(*****
Doel: Deze functie heeft als doel de afstand tussen twee punten te berekenen
Parameters:
real x1			real y1			real x2			real y2
Return value:
real
*****)

Afstand_Punt_Punt := SQRT(((X2-X1)*(X2-X1))+((Y2-Y1)*(Y2-Y1)));
END_FUNCTION

(* Visualisation NavSof
2 more shapes without text or variables
*)
